FUNCTION S8 : INT
VAR_INPUT
    b : USINT;
END_VAR

IF b > 127 THEN
    S8 := USINT_TO_INT(b) - 256;
ELSE
    S8 := USINT_TO_INT(b);
END_IF

END_FUNCTION

(* stored: Version 1.1.0.1
   POU S8: Id {dc4fd68f-ce8c-4c83-b22f-6531310e1c0d}, SpecialFunc None *)
